PROGRAM MAIN
VAR
END_VAR

RilevamentoVeicolo();
MovimentazionePorta();
GestioneChiusura();

ACTION GestioneChiusura:
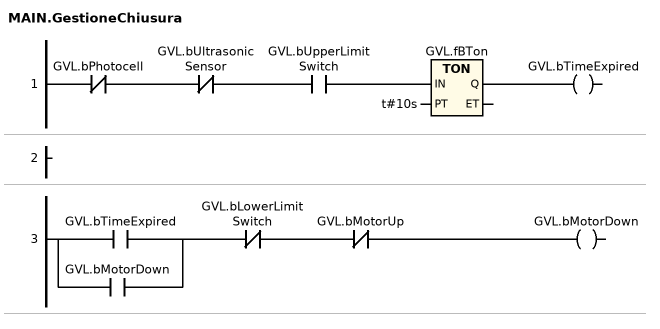
// NETWORK 1
GVL.fBTon(IN := NOT GVL.bPhotocell AND NOT GVL.bUltrasonicSensor AND GVL.bUpperLimitSwitch, PT := t#10s); // TON
GVL.bTimeExpired := GVL.fBTon.Q;

// NETWORK 2

// NETWORK 3
GVL.bMotorDown := (GVL.bTimeExpired OR GVL.bMotorDown) AND NOT GVL.bLowerLimitSwitch AND NOT GVL.bMotorUp;
END_ACTION

ACTION MovimentazionePorta:
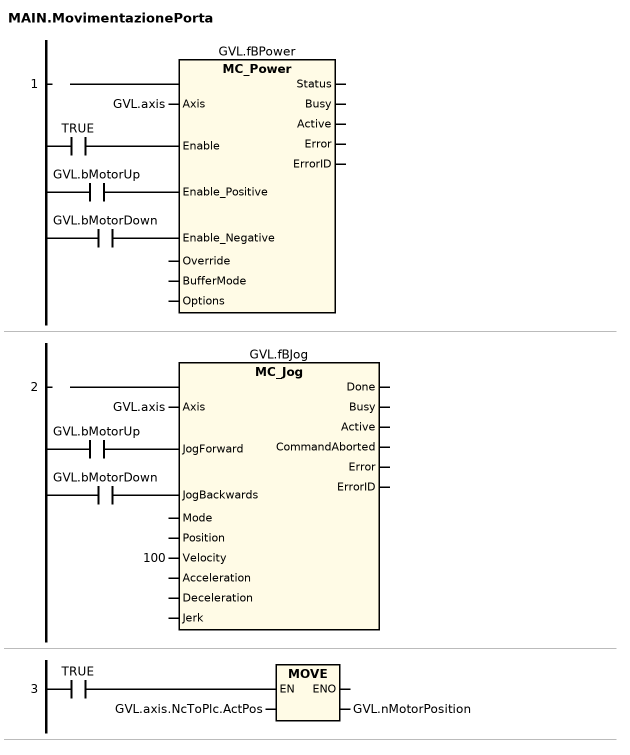
// NETWORK 1
GVL.fBPower(
    Axis := GVL.axis,
    Enable := TRUE,
    Enable_Positive := GVL.bMotorUp,
    Enable_Negative := GVL.bMotorDown); // MC_Power

// NETWORK 2
GVL.fBJog(Axis := GVL.axis, JogForward := GVL.bMotorUp, JogBackwards := GVL.bMotorDown, Velocity := 100); // MC_Jog

// NETWORK 3
GVL.nMotorPosition := GVL.axis.NcToPlc.ActPos;
END_ACTION

ACTION RilevamentoVeicolo:
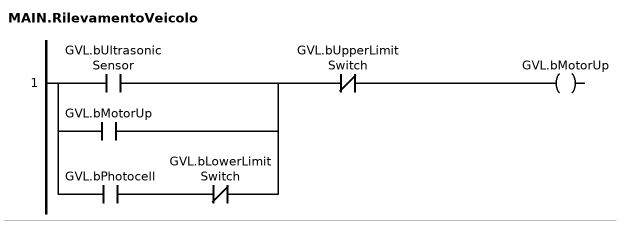
// NETWORK 1
GVL.bMotorUp := (GVL.bUltrasonicSensor OR GVL.bMotorUp OR GVL.bPhotocell AND NOT GVL.bLowerLimitSwitch) AND NOT GVL.bUpperLimitSwitch;
END_ACTION

END_PROGRAM

(* stored: Version 1.1.0.1, ProductVersion 3.1.4024.12
   POU MAIN: Id {f15a0d18-3609-45db-8199-b71f90c9c6f3}, SpecialFunc None
   Action GestioneChiusura: Id {02d9f903-c810-41e8-866f-a20b78e25a48}
   Action MovimentazionePorta: Id {097a3c3a-5458-406a-9471-0adcefc77b8a}
   Action RilevamentoVeicolo: Id {58a29216-9b6a-4898-a724-3758db858095} *)
